{attribute 'GeneratedUsingTerminal: KL9110'}
{attribute addProperty BoxType "KL9110"}
{attribute addProperty Id "PowerAT %I*BOOL0ShortCircuitAT %I*BOOL0"}
{attribute addProperty CRC "1688914119"}
{attribute addProperty Size "0"}
TYPE Channel_64AAC8C7 :
STRUCT
	{attribute addProperty Name "Power"}
	Power AT %I* : BOOL;
	{attribute addProperty Name "ShortCircuit"}
	ShortCircuit AT %I* : BOOL;
END_STRUCT
END_TYPE

(* stored: Version 1.2.0.0, ProductVersion 3.1.4024.9
   DUT Channel_64AAC8C7: Id {0b488639-0781-4611-aeca-77a0161e9865} *)
